PROGRAM DMXTest
VAR
	xConfigSet					: BOOL;
	xStatTestInProgress			: BOOL;
	xDMXSeqTestInProgressOnce	: BOOL;
	xDMXSeqTestInProgressTwice	: BOOL;
	xDMXSeqTestInProgressOnceDC	: BOOL;
	uiCounter2					: UINT;
	uiCounter3					: UINT;
	uiCounter4					: UINT;
	uiCounter5					: UINT;
	uiCounter6					: UINT;
	uiCounter7					: UINT;
	uiCounter8					: UINT;
	uiCounter9					: UINT;
	uiDedicatedRcvdRTIndex		: UINT;
	uiContinuousRTIndex			: UINT;
	
	uiForLoopCfgIndex			: UINT;
//	uiForLoopCtrlWriteIndex		: UINT;
//	uiForLoopCtrlWriteIndex2	: UINT;	
	uiLoopExpctdIndex			: UINT;
	uiForLoopClearExpctd		: UINT;
	uiLoopRcvIndex				: UINT;
	uiByteIndex					: UINT;
	iForLoopRecipeFindMin		: INT;
	iForLoopRecipeFindMax		: INT;
	iForLoopRecipeFindMax1		: INT;
	iForLoopRecipeMin			: INT;
	uiForLoopRecipe				: UINT;
	uiLoopIterDMXDUTArraySeq	: UINT;
	uiLoopIterDMXDUTArrayM		: UINT;
	uiLoopIterDUTArray24V		: UINT;
	uiLoopIterDUTArrayGND		: UINT;
	uiLoopIterTestArrSeq		: UINT;
	uiLoopIterTestArrM			: UINT;
	uiLoopIterTestArr24V		: UINT;
	uiLoopIterTestArrGND		: UINT;	
	iCompareStaticSM			: INT;
	iCompareSeq					: ARRAY[0..ENUM_SeqSM.Twice] OF INT;
	iParseFile					: INT;
	iSetConfig					: INT;
	iSetExpctdBufferSM			: INT;
	iReindexExpctedBufferSM		: INT;
	rt_RunStaticTest			: R_TRIG;
	rt_RunSeqTestOnce			: R_TRIG;
	rt_RunSeqTestOnceDC			: R_TRIG;
	rt_RunSeqTestTwice			: R_TRIG;
	rt_ResetTest				: R_TRIG;
	rt_ResetTestSeq				: R_TRIG;
	rt_ResetTestSeqDC			: R_TRIG;
	r_tStaticTestDone			: R_TRIG;
	
	//Arrays (Refactor 30-09-21)
	arr_uiRecipeIndexTmp		: ARRAY[0..gc.uiDUTConfigCountSplit] OF UINT;
 	arruiDMXChDUTTmp			: ARRAY[0..gc.uiDUTConfigCountSplit] OF UINT;
	arrsDUTChTypeTmp			: ARRAY[0..gc.uiDUTConfigCountSplit] OF STRING[3];	
	arr_uiRecipeIndex			: ARRAY[0..gc.uiDUTConfigCountSplit] OF UINT;
 	arruiDMXChDUT				: ARRAY[0..gc.uiDUTConfigCountSplit] OF UINT;
	arrsDUTChType				: ARRAY[0..gc.uiDUTConfigCountSplit] OF STRING[3];
	xFileImported				: BOOL;
	arr_usiRecipeSettingTmp		: ARRAY[0..gc.uiMaxNrOfDMXChannel] OF USINT;
	arr_usiRecipeSetting		: ARRAY[0..gc.uiMaxNrOfDMXChannel] OF USINT;






	
		
	arrxRcvdBufferPNP24V		: ARRAY[0..gc.uiMaxNrDMXTestCh] OF BOOL;
	arrxRcvdBufferNPN24V		: ARRAY[0..gc.uiMaxNrDMXTestCh] OF BOOL;
	arrxRcvdBufferPNPGND		: ARRAY[0..gc.uiMaxNrDMXTestCh] OF BOOL;
	arrxRcvdBufferNPNGND		: ARRAY[0..gc.uiMaxNrDMXTestCh] OF BOOL;
	
	arrxRcvdBufferPNPSeq		: ARRAY[0..gc.uiMaxNrDMXTestCh] OF BOOL;
	arrxRcvdBufferNPNSeq		: ARRAY[0..gc.uiMaxNrDMXTestCh] OF BOOL;	
	arrxRcvdBufferPNPMotor		: ARRAY[0..gc.uiMaxNrDMXTestCh] OF BOOL;
	arrxRcvdBufferNPNMotor		: ARRAY[0..gc.uiMaxNrDMXTestCh] OF BOOL;
	
	arrxExpctdPNP				: ARRAY[0..gc.uiMaxNrOfDMXChannel] OF BOOL; //What is expected based on the recipe file
	arrxExpctdNPN				: ARRAY[0..gc.uiMaxNrOfDMXChannel] OF BOOL; //What is expected based on the recipe file
	arrxExpctdTmpPNP			: ARRAY[0..gc.uiMaxNrOfDMXChannel] OF BOOL; //What is expected based on the recipe file, reindexed from DUT (usually 0)
	arrxExpctdTmpNPN			: ARRAY[0..gc.uiMaxNrOfDMXChannel] OF BOOL; //What is expected based on the recipe file, reindexed from DUT (usually 0)
	arrxExpctdTmpPNP24V			: ARRAY[0..gc.uiMaxNrDMXTestCh] OF BOOL; //What is expected based on the recipe file, reindexed from DUT (usually 0)
	arrxExpctdTmpNPN24V			: ARRAY[0..gc.uiMaxNrDMXTestCh] OF BOOL; //What is expected based on the recipe file, reindexed from DUT (usually 0)
	arrxExpctdTmpPNPGND			: ARRAY[0..gc.uiMaxNrDMXTestCh] OF BOOL; //What is expected based on the recipe file, reindexed from DUT (usually 0)
	arrxExpctdTmpNPNGND			: ARRAY[0..gc.uiMaxNrDMXTestCh] OF BOOL; //What is expected based on the recipe file, reindexed from DUT (usually 0)

	arrxExpctdTmpPNPSeqDMX		: ARRAY[0..gc.uiMaxNrDMXTestCh] OF BOOL; //What is expected based on the recipe file, reindexed from DUT (usually 0)
	arrxExpctdTmpNPNSeqDMX		: ARRAY[0..gc.uiMaxNrDMXTestCh] OF BOOL; //What is expected based on the recipe file, reindexed from DUT (usually 0)
	arrxExpctdTmpPNPSeqDC		: ARRAY[0..gc.uiMaxNrDMXTestCh] OF BOOL; //What is expected based on the recipe file, reindexed from DUT (usually 0)
	arrxExpctdTmpNPNSeqDC		: ARRAY[0..gc.uiMaxNrDMXTestCh] OF BOOL; //What is expected based on the recipe file, reindexed from DUT (usually 0)

	arrxExpctdTmpPNPSeq			: ARRAY[0..gc.uiMaxNrOfDMXChannel] OF BOOL; //What is expected based on the recipe file, reindexed from DUT (usually 0)
	arrxExpctdTmpNPNSeq			: ARRAY[0..gc.uiMaxNrOfDMXChannel] OF BOOL; //What is expected based on the recipe file, reindexed from DUT (usually 0)
	arrxExpctdTmpPNPMotor		: ARRAY[0..gc.uiMaxNrOfDMXChannel] OF BOOL; //What is expected based on the recipe file, reindexed from DUT (usually 0)
	arrxExpctdTmpNPNMotor		: ARRAY[0..gc.uiMaxNrOfDMXChannel] OF BOOL; //What is expected based on the recipe file, reindexed from DUT (usually 0)
	
	arrxExpctdMaskPNPSeq		: ARRAY[0..gc.uiMaxNrOfDMXChannel] OF BOOL; //Copy the contents of hardware buffer 
	arrxExpctdMaskNPNSeq		: ARRAY[0..gc.uiMaxNrOfDMXChannel] OF BOOL; //Copy the contents of hardware buffer 
	arr_diTestStaticPNP24V		: ARRAY[0..gc.uiMaxNrDMXTestCh] OF DINT;
	arr_diTestStaticNPN24V		: ARRAY[0..gc.uiMaxNrDMXTestCh] OF DINT;
	arr_diTestStaticPNPGND		: ARRAY[0..gc.uiMaxNrDMXTestCh] OF DINT;
	arr_diTestStaticNPNGND		: ARRAY[0..gc.uiMaxNrDMXTestCh] OF DINT;
	arr_diTestPNPSeqOnceLine			: ARRAY[0..gc.uiMaxNrDMXTestCh] OF DINT;
	arr_diTestPNPSeqOnceLineTmp			: ARRAY[0..gc.uiMaxNrDMXTestCh] OF DINT;
	arr_diTestNPNSeqOnceLine			: ARRAY[0..gc.uiMaxNrDMXTestCh] OF DINT;
	arr_diTestNPNSeqOnceLineTmp			: ARRAY[0..gc.uiMaxNrDMXTestCh] OF DINT;

	arr_udiMEMCPYPNPSeqOnceRcvdTmp		: ARRAY[0..gc.uiMaxNrDMXTestCh] OF UDINT;
	arr_udiMEMCPYNPNSeqOnceRcvdTmp		: ARRAY[0..gc.uiMaxNrDMXTestCh] OF UDINT;
			
	diTestStaticPNP24V				: DINT;
	diTestStaticNPN24V				: DINT;
	diTestStaticPNPGND				: DINT;	
	diTestStaticNPNGND				: DINT;
	
	diTestPNPSeqOnceComplete		: DINT;

	arrdiTestPNPSeqOnceComplete		: ARRAY[0..gc.uiMaxNrDMXTestCh] OF DINT;
	arrdiTestPNPSeqOnceCompleteTmp	: ARRAY[0..gc.uiMaxNrDMXTestCh] OF DINT;

	arrdiTestNPNSeqOnceComplete		: ARRAY[0..gc.uiMaxNrDMXTestCh] OF DINT;
	arrdiTestNPNSeqOnceCompleteTmp	: ARRAY[0..gc.uiMaxNrDMXTestCh] OF DINT;

	arrdiTestNPNSeqOnceCompleteProblemIndex		: ARRAY[0..gc.uiMaxNrDMXTestCh] OF DINT;
	
	arrudiStaticCopyResultPNP24V	: ARRAY[0..gc.uiMaxNrOfDMXChannel] OF UDINT;
	arrudiStaticCopyResultNPN24V	: ARRAY[0..gc.uiMaxNrOfDMXChannel] OF UDINT;
	arrudiStaticCopyResultPNPGND	: ARRAY[0..gc.uiMaxNrOfDMXChannel] OF UDINT;
	arrudiStaticCopyResultNPNGND	: ARRAY[0..gc.uiMaxNrOfDMXChannel] OF UDINT;	

	arr_diTestPNPMotorDir1		: ARRAY[0..gc.uiMaxNrDMXTestCh] OF DINT;
	arr_diTestNPNMotorDir1		: ARRAY[0..gc.uiMaxNrDMXTestCh] OF DINT;
	arr_diTestPNPMotorDir2		: ARRAY[0..gc.uiMaxNrDMXTestCh] OF DINT;
	arr_diTestNPNMotorDir2		: ARRAY[0..gc.uiMaxNrDMXTestCh] OF DINT;

	
	
	diCompTestResult			: DINT;
	diCompTestResultTemp		: DINT;
	diTestResultStaticPNP		: DINT;
	diTestResultStaticNPN		: DINT;	

	arrVisu_diTestResult		: ARRAY[0..gc.uiMaxNrDMXTestCh] OF DINT;
	uiVisuIndex					: UINT;
	tonReadWait					: TON;
	tonConvert					: TON;
	tonWriteCopyWait			: TON;
	tonTestIterGap				: TON;
	tTestTime					: TIME;
	tWriteWaitTime				: TIME;
	r_tSetConfig				: R_TRIG;
	uiRecipeIndexRcv			: UINT;
	uiMinRecipeIndex			: UINT;
	uiMaxRecipeIndex			: UINT;
	cuiMinDUTIndex				: UINT	:= 0; // Constant
	uiMaxRecipeIndexTemp		: UINT;
	arruiMotorTestIndices		: ARRAY[0..gc.uiMaxNrOfDMXChannel] OF UINT;
	arruiMotorTestIndicesTmp	: ARRAY[0..gc.uiMaxNrOfDMXChannel] OF UINT;
	arruiSeqTestIndices			: ARRAY[0..gc.uiMaxNrOfDMXChannel] OF UINT;
	arruiSeqTestIndicesTmp		: ARRAY[0..gc.uiMaxNrOfDMXChannel] OF UINT;
	
	arruiSeqTestIndicesDMX			: ARRAY[0..gc.uiMaxNrDMXTestCh] OF UINT;
	arruiSeqTestIndicesDMXSW		: ARRAY[0..gc.uiMaxNrDMXTestCh] OF UINT;
	arruiSeqTestIndicesDMXTmp		: ARRAY[0..gc.uiMaxNrDMXTestCh] OF UINT;
	
	arruiSeqTestIndicesDC			: ARRAY[0..gc.uiMaxNrDMXTestCh] OF UINT;
	arruiSeqTestIndicesDCTmp		: ARRAY[0..gc.uiMaxNrDMXTestCh] OF UINT;	
	
	arrui24VTestIndices			: ARRAY[0..gc.uiMaxNrOfDMXChannel] OF UINT;
	arrui24VTestIndicesTmp		: ARRAY[0..gc.uiMaxNrOfDMXChannel] OF UINT;
	arruiGNDTestIndices			: ARRAY[0..gc.uiMaxNrOfDMXChannel] OF UINT;
	arruiGNDTestIndicesTmp		: ARRAY[0..gc.uiMaxNrOfDMXChannel] OF UINT;
	udiMemCpyResultPNP			: UDINT;
	udiMemCpyResultDMX			: UDINT;	
	r_tSetExpectedBuff			: R_TRIG;
	r_tExpectedBufferSet		: R_TRIG;
	uiLoopExpctdIndexRead		: UINT;
	uiLoopExpctdIndexWrite		: UINT;
	xTestBoolDelete				: BOOL;
	uiForLoopZeroStorageArray	: UINT;
	
	//For DUT Config
	r_tSetDUTVal				: R_TRIG;
	usiDUTVal					: USINT;
	uiForLoopDUTIter			: UINT;
	iSetDUTSM					: INT;
	
	//For 'Invert Recipe Settings'
	uiStartingIndex				: UINT;
	uiEndingIndex				: UINT;
	uiRecipeInvertIter			: UINT;
	R_TInvertRecipe				: R_TRIG;
	iInvertRecipeSM				: INT;
END_VAR

SeqTestOnce();
//SeqTestTwice();
//SeqTestOnceDC();
InvertRecipeSettings();
rt_RunStaticTest();
rt_ResetTest();
r_tSetConfig();//Set config when file is loaded; this condition happens when End-of-File (EOF) is reached; set by HMI button
r_tSetExpectedBuff(CLK:=r_tSetConfig.Q);
r_tExpectedBufferSet();
r_tStaticTestDone(CLK			:= (iCompareStaticSM = 110));
r_tSetDUTVal();
tonReadWait(PT		:= tTestTime);
tonConvert(PT		:= tTestTime);
tonWriteCopyWait(PT	:= tWriteWaitTime);
tonTestIterGap(PT	:= tTestTime);
tTestTime			:= T#80MS;
//just an example one
tWriteWaitTime		:= T#10MS; // same as the tOffDelay set to the input debounce FB
//DMX DUT Channels, Software 0-255 
//DMX Config Channels, Software, 256-511
//DMX DUT Channels, Hardware 1-256
//DMX Config Channels, Hardware, 257-512

//Interface Link - continued - DMXTest Local Vars

//"Config Complete" Expctd Buffer, and "Config Complete" Received Buffer; then Global Comparison is like 'masking' all but one channel at a time;

CASE iParseFile OF

0:
IF P_TextModeRead.r_tFileChg.Q THEN
	xFileImported		:= FALSE;	
	iParseFile			:= 5;
END_IF

5:
IF P_TextModeRead.fbFileGets.bEOF THEN
	uiForLoopRecipe	:= 0; // Reset the iterator used in the next state of the SM
	iParseFile		:= 10;
END_IF
	
10://At first check for any recipe items specified in the file;
//Load the recipe data into respective arrays
//For recipe indices = 0 to 255, parse the file to read the recipe index, DMX channel, and channel type
FOR uiForLoopRecipe := 0 TO gc.uiDUTConfigCountSplit BY 1 DO
	//Read the Recipe Index
	arr_uiRecipeIndexTmp[uiForLoopRecipe]		:= STRING_TO_UINT(P_TextModeRead.database[uiForLoopRecipe,0]);
	//Read the DMX Channel for the DUT
	arruiDMXChDUTTmp[uiForLoopRecipe]			:= STRING_TO_UINT(P_TextModeRead.database[uiForLoopRecipe,1]);
	//Read the type of Channel on the DUT
	arrsDUTChTypeTmp[uiForLoopRecipe]			:= P_TextModeRead.database[uiForLoopRecipe,2];
END_FOR
//Stash the values from temp (inside FOR loop) to other arrays
arr_uiRecipeIndex	:= arr_uiRecipeIndexTmp;
arruiDMXChDUT		:= arruiDMXChDUTTmp;
arrsDUTChType		:= arrsDUTChTypeTmp;

//If the 'TextModeRead' re-enters 'Ready' state then advance this SM
IF P_TextModeRead.step = 0 THEN
	xFileImported		:= TRUE;
	iParseFile			:= 0;	
END_IF

END_CASE

CASE iSetConfig OF

//Don't look at the P_TextRead; evaluate on the arrays you just imported

0:
IF r_tSetConfig.Q THEN
	iSetConfig			:= 10;	
END_IF

10://Read the string that is loaded from file reader; pass value to DMX Function Block, at the appropriate Config index
//This is the setting to control the position of the 'config' relays on the tester
//Ensure that the declared arrays are sufficiently long to handle the max conceivable value (512 x 2, in this case?)
FOR uiForLoopRecipe := 0 TO gc.uiDUTConfigCountSplit BY 1 DO
	IF (arruiDMXChDUT[uiForLoopRecipe] <> 0) THEN
		//Set the config routing := NPN
		arr_usiRecipeSettingTmp[(uiForLoopRecipe+gc.uiChannelSplitCount)]	:= 255;
	ELSIF (arruiDMXChDUT[uiForLoopRecipe] = 0) THEN
		//Set the config routing := PNP
		arr_usiRecipeSettingTmp[(uiForLoopRecipe+gc.uiChannelSplitCount)]	:= 0;
	END_IF	
END_FOR
//Stash the values from temp (inside FOR loop) to other arrays
arr_usiRecipeSetting	:= arr_usiRecipeSettingTmp;

	iSetConfig			:= 20;	

20://Iterate over the config listings to create indices for what must be tested static (power, ground), and what must be tested sequentially (channels)
uiLoopIterDMXDUTArraySeq	:= 0;
uiLoopIterTestArrSeq		:= 0;
//Zero out the array that is copied to in the next state of the SM
FOR uiForLoopZeroStorageArray	:= 0 TO gc.uiMaxNrOfDMXChannel BY 1 DO
	arruiSeqTestIndicesTmp[uiForLoopZeroStorageArray]	:= 0;
END_FOR
//Stash the values from temp (inside FOR loop) to other arrays
arruiSeqTestIndices		:= arruiSeqTestIndicesTmp;
iSetConfig				:= 40;	

40:
//For any 'DMX'-type channels with an assigned channel # (from the recipe), then copy only those elements to another array
//These are elements that are tested sequentially - once - so this includes Dry Contacts but not Motors
REPEAT
	IF ((arrsDUTChType[uiLoopIterDMXDUTArraySeq] = 'DMX') OR (arrsDUTChType[uiLoopIterDMXDUTArraySeq] = '24V')) AND (arruiDMXChDUT[uiLoopIterDMXDUTArraySeq] <> 0) THEN
		MEMCPY(srcAddr:=ADR(arruiDMXChDUT[uiLoopIterDMXDUTArraySeq]),destAddr:=ADR(arruiSeqTestIndicesTmp[uiLoopIterDMXDUTArraySeq]),n:=SIZEOF(arruiDMXChDUT[uiLoopIterDMXDUTArraySeq])); //UINT = 4 bytes?
//		uiLoopIterTestArrSeq		:= uiLoopIterTestArrSeq+1;
	END_IF
	uiLoopIterDMXDUTArraySeq	:= uiLoopIterDMXDUTArraySeq+1;
UNTIL 
(uiLoopIterDMXDUTArraySeq = gc.uiMaxNrOfDMXChannel)
END_REPEAT
//Stash the values from temp (inside FOR loop) to other arrays
arruiSeqTestIndices		:= arruiSeqTestIndicesTmp;

iSetConfig					:= 50;	

50:
//Use different iterators - set them to 0 prior to use
uiLoopIterDMXDUTArrayM		:= 0;
uiLoopIterTestArrM			:= 0;
//Zero out the array that is copied to in the next state of the SM
FOR uiForLoopZeroStorageArray	:= 0 TO gc.uiMaxNrOfDMXChannel BY 1 DO
	arruiMotorTestIndicesTmp[uiForLoopZeroStorageArray]	:= 0;
END_FOR
//Stash the values from temp (inside FOR loop) to other arrays
arruiMotorTestIndices	:= arruiMotorTestIndicesTmp;

iSetConfig					:= 60;	

60:
//Motors - Type code "M" - must be tested both in the PNP & NPN inputs
//This array easily provides the indexing for which channels the motors are on
REPEAT
	IF (arrsDUTChType[uiLoopIterDMXDUTArrayM] = 'M') AND (arruiDMXChDUT[uiLoopIterDMXDUTArrayM] <> 0)  THEN
		MEMCPY(srcAddr:=ADR(arruiDMXChDUT[uiLoopIterDMXDUTArrayM]),destAddr:=ADR(arruiMotorTestIndicesTmp[uiLoopIterDMXDUTArrayM]),n:=SIZEOF(arruiDMXChDUT[uiLoopIterDMXDUTArrayM])); //UINT = 4 bytes?
//		uiLoopIterTestArrM		:= uiLoopIterTestArrM+1;
	END_IF
	uiLoopIterDMXDUTArrayM	:= uiLoopIterDMXDUTArrayM+1;
UNTIL 
(uiLoopIterDMXDUTArrayM = gc.uiMaxNrOfDMXChannel)
END_REPEAT
//Stash the values from temp (inside FOR loop) to other arrays
arruiMotorTestIndices	:= arruiMotorTestIndicesTmp;

iSetConfig		:= 70;

70:
//Use different iterators - set them to 0 prior to use
uiLoopIterDUTArray24V		:= 0;
uiLoopIterTestArr24V		:= 0;
//Zero out the array that is copied to in the next state of the SM
FOR uiForLoopZeroStorageArray	:= 0 TO gc.uiMaxNrOfDMXChannel BY 1 DO
	arrui24VTestIndicesTmp[uiForLoopZeroStorageArray]	:= 0;
END_FOR
//Stash the values from temp (inside FOR loop) to other arrays
arrui24VTestIndices		:= arrui24VTestIndicesTmp;

iSetConfig				:= 80;

80:
//24V - Type code "24V" - is tested per static config
//This array easily provides the indexing for which channels the 24V are on
REPEAT
	IF (arrsDUTChType[uiLoopIterDUTArray24V] = '24V') AND (arruiDMXChDUT[uiLoopIterDUTArray24V] = 0) THEN
		MEMCPY(srcAddr:=ADR(arr_uiRecipeIndex[uiLoopIterDUTArray24V]),destAddr:=ADR(arrui24VTestIndicesTmp[uiLoopIterDUTArray24V]),n:=SIZEOF(arr_uiRecipeIndex[uiLoopIterDUTArray24V])); //UINT = 2 bytes?
//		uiLoopIterTestArr24V	:= uiLoopIterTestArr24V +1;
	END_IF
	uiLoopIterDUTArray24V	:= uiLoopIterDUTArray24V+1;
UNTIL 
(uiLoopIterDUTArray24V = gc.uiDUTConfigCountSplit)
END_REPEAT
//Stash the values from temp (inside FOR loop) to other arrays
arrui24VTestIndices	:= arrui24VTestIndicesTmp;

iSetConfig		:= 90;

90://Clear Iterators for GND channel indexing
//Use different iterators - set them to 0 prior to use
uiLoopIterDUTArrayGND		:= 0;
uiLoopIterTestArrGND		:= 0;
//Zero out the array that is copied to in the next state of the SM
FOR uiForLoopZeroStorageArray	:= 0 TO gc.uiMaxNrOfDMXChannel BY 1 DO
	arruiGNDTestIndicesTmp[uiForLoopZeroStorageArray]	:= 0;
END_FOR
//Stash the values from temp (inside FOR loop) to other arrays
arruiGNDTestIndices		:= arruiGNDTestIndicesTmp;

iSetConfig				:= 100;

100:
//Ground - Type code "GND" - is tested per static config
//This array easily provides the indexing for which channels the 24V are on
REPEAT
	IF (arrsDUTChType[uiLoopIterDUTArrayGND] = 'GND') AND (arruiDMXChDUT[uiLoopIterDUTArrayGND] = 0) THEN
		MEMCPY(srcAddr:=ADR(arr_uiRecipeIndex[uiLoopIterDUTArrayGND]),destAddr:=ADR(arruiGNDTestIndicesTmp[uiLoopIterDUTArrayGND]),n:=SIZEOF(arr_uiRecipeIndex[uiLoopIterDUTArrayGND])); //UINT = 4 bytes?
//		uiLoopIterTestArrGND	:= uiLoopIterTestArrGND+1;
	END_IF
	uiLoopIterDUTArrayGND	:= uiLoopIterDUTArrayGND+1;
UNTIL 
(uiLoopIterDUTArrayGND = gc.uiDUTConfigCountSplit)
END_REPEAT
//Stash the values from temp (inside FOR loop) to other arrays
arruiGNDTestIndices	:= arruiGNDTestIndicesTmp;

iSetConfig				:= 110;

//Copy of state30
110://Iterate over the config listings to create indices for what must be tested static (power, ground), and what must be tested sequentially (channels)
uiLoopIterDMXDUTArraySeq		:= 0;
uiLoopIterTestArrSeq			:= 0;
//Zero out the array that is copied to in the next state of the SM
FOR uiForLoopZeroStorageArray	:= 0 TO gc.uiMaxNrOfDMXChannel BY 1 DO
	arruiSeqTestIndicesDMXTmp[uiForLoopZeroStorageArray]	:= 0;
	arruiSeqTestIndicesDMXSW[uiForLoopZeroStorageArray]		:= 0;
END_FOR
//Stash the values from temp (inside FOR loop) to other arrays
arruiSeqTestIndicesDMX			:= arruiSeqTestIndicesDMXTmp;
iSetConfig						:= 120;	

120://Effectively a copy of state40
//For any 'DMX'-type channels with an assigned channel # (from the recipe), then copy only those elements to another array
//These are elements that are tested sequentially - once - so this includes Dry Contacts but not Motors
REPEAT
	IF (arrsDUTChType[uiLoopIterDMXDUTArraySeq] = 'DMX') AND (arruiDMXChDUT[uiLoopIterDMXDUTArraySeq] <> 0) THEN
		MEMCPY(srcAddr:=ADR(arruiDMXChDUT[uiLoopIterDMXDUTArraySeq]),destAddr:=ADR(arruiSeqTestIndicesDMXTmp[uiLoopIterDMXDUTArraySeq]),n:=SIZEOF(arr_uiRecipeIndex[uiLoopIterDUTArrayGND])); //UINT = 4 bytes?
//		uiLoopIterTestArrSeq		:= uiLoopIterTestArrSeq+1;
	END_IF
	uiLoopIterDMXDUTArraySeq		:= uiLoopIterDMXDUTArraySeq+1;
UNTIL 
(uiLoopIterDMXDUTArraySeq = gc.uiMaxNrOfDMXChannel)
END_REPEAT
//Stash the values from temp (inside FOR loop) to other arrays
arruiSeqTestIndicesDMX				:= arruiSeqTestIndicesDMXTmp;

//Set the recipe addresses one lower for 'SW'-Software-because software indexes from 0, not 1
FOR uiCounter8	:= 0 TO gc.uiMaxNrDMXTestCh BY 1 DO
	IF arruiSeqTestIndicesDMX[uiCounter8] <> 0 THEN
		arruiSeqTestIndicesDMXSW[uiCounter8]	:= arruiSeqTestIndicesDMX[uiCounter8] - 1;	
	END_IF
END_FOR

iSetConfig							:= 130;	

//Copy of state30
130://Iterate over the config listings to create indices for what must be tested static (power, ground), and what must be tested sequentially (channels)
uiLoopIterDMXDUTArraySeq		:= 0;
uiLoopIterTestArrSeq			:= 0;
//Zero out the array that is copied to in the next state of the SM
FOR uiForLoopZeroStorageArray	:= 0 TO gc.uiMaxNrOfDMXChannel BY 1 DO
	arruiSeqTestIndicesDCTmp[uiForLoopZeroStorageArray]	:= 0;
END_FOR
//Stash the values from temp (inside FOR loop) to other arrays
arruiSeqTestIndicesDC			:= arruiSeqTestIndicesDCTmp;
iSetConfig						:= 140;	

140:
//For any 'DMX'-type channels with an assigned channel # (from the recipe), then copy only those elements to another array
//These are elements that are tested sequentially - once - so this includes Dry Contacts but not Motors
REPEAT
	IF (arrsDUTChType[uiLoopIterDMXDUTArraySeq] = '24V') AND (arruiDMXChDUT[uiLoopIterDMXDUTArraySeq] <> 0) THEN
		MEMCPY(srcAddr:=ADR(arruiDMXChDUT[uiLoopIterDMXDUTArraySeq]),destAddr:=ADR(arruiSeqTestIndicesDCTmp[uiLoopIterDMXDUTArraySeq]),n:=SIZEOF(arruiDMXChDUT[uiLoopIterDMXDUTArraySeq])); //UINT = 4 bytes?
//		uiLoopIterTestArrSeq		:= uiLoopIterTestArrSeq+1;
	END_IF
	uiLoopIterDMXDUTArraySeq		:= uiLoopIterDMXDUTArraySeq+1;
UNTIL 
(uiLoopIterDMXDUTArraySeq = gc.uiMaxNrOfDMXChannel)
END_REPEAT
//Stash the values from temp (inside FOR loop) to other arrays
arruiSeqTestIndicesDC				:= arruiSeqTestIndicesDCTmp;

iSetConfig							:= 0;	

END_CASE


//Set the config of the 'routing' channels
IF r_tSetConfig.Q THEN
	g_ast.DMXHWOut	:= g_ast.DMXPhysOut;
//	xConfigSet		:= TRUE;
END_IF


// For manual setting of channels from the Visualization - NOTE! This stamps over any other values set for the lower 256 channels (DUT)
CASE iSetDUTSM OF
	
0:
IF r_tSetDUTVal.Q THEN
	iSetDUTSM		:= 10;
END_IF

10:
FOR uiForLoopDUTIter := 0 TO gc.uiDUTConfigCountSplit BY 1 DO
	g_ast.DMXHWOut[uiForLoopDUTIter] 	:= usiDUTVal;
END_FOR
//g_ast.DMXHWOut					:= g_ast.DMXPhysOut;

IF NOT r_tSetDUTVal.Q THEN
	iSetDUTSM	:= 0;
END_IF

END_CASE


CASE iSetExpctdBufferSM OF
	
0://If there is a trigger to set the test config, create a new 'Expctd' buffer
IF r_tSetExpectedBuff.Q THEN
	r_tExpectedBufferSet.CLK	:= FALSE;
	//Clear the existing buffers
	FOR uiForLoopClearExpctd := 0 TO gc.uiMaxNrOfDMXChannel BY 1 DO
		arrxExpctdPNP[uiForLoopClearExpctd]	:= 0;
		arrxExpctdNPN[uiForLoopClearExpctd]	:= 0;
	END_FOR
	iSetExpctdBufferSM			:= 10;
END_IF

10: // Set Expected Buffers per Recipe Files
FOR uiLoopExpctdIndex := 0 TO gc.uiMaxNrOfDMXChannel BY 1 DO
	IF (arr_usiRecipeSetting[uiLoopExpctdIndex] <= 127) THEN
		arrxExpctdPNP[arr_uiRecipeIndex[uiLoopExpctdIndex]]		:= TRUE; 
		arrxExpctdNPN[arr_uiRecipeIndex[uiLoopExpctdIndex]]		:= FALSE;
	ELSIF (arr_usiRecipeSetting[uiLoopExpctdIndex] > 127) THEN
		arrxExpctdPNP[arr_uiRecipeIndex[uiLoopExpctdIndex]]		:= FALSE;
		arrxExpctdNPN[arr_uiRecipeIndex[uiLoopExpctdIndex]]		:= TRUE; 
	END_IF
	//Zero out Expected, type-specific index buffers
	arrxExpctdTmpPNP24V[uiLoopExpctdIndex] 					:= 0;
	arrxExpctdTmpNPN24V[uiLoopExpctdIndex] 					:= 0;
	arrxExpctdTmpPNPGND[uiLoopExpctdIndex] 					:= 0;
	arrxExpctdTmpNPNGND[uiLoopExpctdIndex] 					:= 0;
END_FOR

r_tExpectedBufferSet.CLK	:= TRUE;
iSetExpctdBufferSM			:= 0;

END_CASE

CASE iReindexExpctedBufferSM OF
	
0:
IF r_tExpectedBufferSet.Q THEN
	iReindexExpctedBufferSM	:= 10;
END_IF

10://Copy the contents of Expected Buffer to a different Buffer, starting at array address 0 - only the channels that have a hardware input index
MEMCPY(srcAddr:=ADR(arrxExpctdPNP[gc.uiChannelSplitCount]),destAddr:=ADR(arrxExpctdTmpPNP[cuiMinDUTIndex]),n:=gc.uiChannelsUT);
MEMCPY(srcAddr:=ADR(arrxExpctdNPN[gc.uiChannelSplitCount]),destAddr:=ADR(arrxExpctdTmpNPN[cuiMinDUTIndex]),n:=gc.uiChannelsUT);

iReindexExpctedBufferSM	:= 20;

20:
//And create the comparison Expected Buffer for Static Test - 24V & GND indices
FOR uiCounter5 := 0 TO gc.uiMaxNrDMXTestCh BY 1 DO
	IF arrui24VTestIndices[uiCounter5] <> 0 THEN	
		MEMCPY(srcAddr:=ADR(arrxExpctdTmpPNP[arrui24VTestIndices[uiCounter5]]),destAddr:=ADR(arrxExpctdTmpPNP24V[arrui24VTestIndices[uiCounter5]]),n:=SIZEOF(arrxExpctdTmpPNP[arrui24VTestIndices[uiCounter5]])); //bytes
		MEMCPY(srcAddr:=ADR(arrxExpctdTmpNPN[arrui24VTestIndices[uiCounter5]]),destAddr:=ADR(arrxExpctdTmpNPN24V[arrui24VTestIndices[uiCounter5]]),n:=SIZEOF(arrxExpctdTmpNPN[arrui24VTestIndices[uiCounter5]])); //bytes
	END_IF
	
	IF arruiGNDTestIndices[uiCounter5] <> 0 THEN	
		MEMCPY(srcAddr:=ADR(arrxExpctdTmpPNP[arruiGNDTestIndices[uiCounter5]]),destAddr:=ADR(arrxExpctdTmpPNPGND[arruiGNDTestIndices[uiCounter5]]),n:=SIZEOF(arrxExpctdTmpPNP[arruiGNDTestIndices[uiCounter5]])); //bytes
		MEMCPY(srcAddr:=ADR(arrxExpctdTmpNPN[arruiGNDTestIndices[uiCounter5]]),destAddr:=ADR(arrxExpctdTmpNPNGND[arruiGNDTestIndices[uiCounter5]]),n:=SIZEOF(arrxExpctdTmpNPN[arruiGNDTestIndices[uiCounter5]])); //bytes
	END_IF	
END_FOR

iReindexExpctedBufferSM	:= 0;

END_CASE


CASE iCompareStaticSM OF
	
0: // If test is triggered by user
IF rt_RunStaticTest.Q THEN
	xStatTestInProgress						:= TRUE;
	uiLoopRcvIndex							:= cuiMinDUTIndex; 
	iCompareStaticSM						:= 10;
END_IF

10: // Zero out all comparison buffers before each comparison
//IF (uiLoopRcvIndex=0) THEN
	IF xStatTestInProgress THEN
		//by default, Counter = 0 at the first initialization; it is reset at the end of this State Machine
		//Clear Storage Buffers pre-test to ensure no old data interferes with current test
		FOR uiCounter4 := 0 TO gc.uiDUTConfigCountSplit BY 1 DO
			arrxRcvdBufferPNP24V[uiCounter4]	:= 0;		
			arrxRcvdBufferNPN24V[uiCounter4]	:= 0;		
			arrxRcvdBufferPNPGND[uiCounter4]	:= 0;		
			arrxRcvdBufferNPNGND[uiCounter4]	:= 0;
			gFB.arrFB_DMX[uiCounter4].I.xCmdOff	:= TRUE;		
//			g_ast.DMX[uiCounter4].IQ.xCmdOff	:= TRUE;	
		END_FOR
	iCompareStaticSM				:= 20;
	END_IF
(*
ELSIF (uiLoopRcvIndex>0) THEN
	IF xStatTestInProgress AND tonTestIterGap.Q THEN
		tonTestIterGap.IN	:= FALSE;
		//by default, Counter = 0 at the first initialization; it is reset at the end of this State Machine
		//Clear Storage Buffers pre-test to ensure no old data interferes with current test
		FOR uiCounter4 := 0 TO gc.uiDUTConfigCountSplit BY 1 DO
			arrxRcvdBufferPNP24V[uiCounter4]	:= 0;		
			arrxRcvdBufferNPN24V[uiCounter4]	:= 0;		
			arrxRcvdBufferPNPGND[uiCounter4]	:= 0;		
			arrxRcvdBufferNPNGND[uiCounter4]	:= 0;		
		END_FOR
	iCompareStaticSM				:= 30; // don't write the hardware value (skip 20)
	END_IF
END_IF
*)
	
20:	
//write 'hardware-clear' state 
g_ast.DMXHWOut					:= g_ast.DMXPhysOut;
iCompareStaticSM				:= 30;

30: //Set the Expected Mask & write data to controller
(*
IF uiLoopRcvIndex <> 0 THEN
//	g_ast.DMX[uiLoopRcvIndex].IQ.xCmdOn			:= TRUE;
	FOR uiCounter3 := cuiMinDUTIndex TO gc.uiMaxNrDMXTestCh BY 1 DO
		IF uiCounter3 <> uiLoopRcvIndex THEN
			g_ast.DMX[uiCounter3].IQ.xCmdOff	:= TRUE;	
		END_IF
	END_FOR
	iCompareStaticSM		:= 40;
ELSE //uiLoopRcvIndex = 0
	*)
tonWriteCopyWait.IN		:= TRUE;
iCompareStaticSM		:= 50;
//END_IF

40:
//Write DMX channels
(*
g_ast.DMXHWOut			:= g_ast.DMXPhysOut;
tonWriteCopyWait.IN		:= TRUE;
iCompareStaticSM		:= 50;
*)

50:
IF tonWriteCopyWait.Q THEN
	tonWriteCopyWait.IN	:= FALSE;
	iCompareStaticSM	:= 60;
END_IF

60:
FOR uiCounter4 := 0 TO gc.uiMaxNrDMXTestCh BY 1 DO

//IF there is an index for a '24V' element, then copy that element's value to a new pair of arrays, for 'Received'

	IF arrui24VTestIndices[uiCounter4] <> 0 THEN

		arrudiStaticCopyResultPNP24V[arrui24VTestIndices[uiCounter4]]	:= MEMCPY(srcAddr:=ADR(g_ast.arrInputPNP[arrui24VTestIndices[uiCounter4]]),destAddr:=ADR(arrxRcvdBufferPNP24V[arrui24VTestIndices[uiCounter4]]),n:=SIZEOF(g_ast.arrInputPNP[arrui24VTestIndices[uiCounter4]])); //bytes
		arrudiStaticCopyResultNPN24V[arrui24VTestIndices[uiCounter4]]	:= MEMCPY(srcAddr:=ADR(g_ast.arrInputNPN[arrui24VTestIndices[uiCounter4]]),destAddr:=ADR(arrxRcvdBufferNPN24V[arrui24VTestIndices[uiCounter4]]),n:=SIZEOF(g_ast.arrInputNPN[arrui24VTestIndices[uiCounter4]])); //bytes)

	END_IF

//IF there is an index for a 'GND' element, then copy that element's value to a new pair of arrays, for 'Received'

	IF arruiGNDTestIndices[uiCounter4] <> 0 THEN

		arrudiStaticCopyResultPNPGND[arruiGNDTestIndices[uiCounter4]]	:= MEMCPY(srcAddr:=ADR(g_ast.arrInputPNP[arruiGNDTestIndices[uiCounter4]]),destAddr:=ADR(arrxRcvdBufferPNPGND[arruiGNDTestIndices[uiCounter4]]),n:=SIZEOF(g_ast.arrInputPNP[arruiGNDTestIndices[uiCounter4]])); //bytes
		arrudiStaticCopyResultNPNGND[arruiGNDTestIndices[uiCounter4]]	:= MEMCPY(srcAddr:=ADR(g_ast.arrInputNPN[arruiGNDTestIndices[uiCounter4]]),destAddr:=ADR(arrxRcvdBufferNPNGND[arruiGNDTestIndices[uiCounter4]]),n:=SIZEOF(g_ast.arrInputNPN[arruiGNDTestIndices[uiCounter4]])); //bytes)
	
	END_IF
	
END_FOR

iCompareStaticSM			:= 70;

70:
tonReadWait.IN				:= TRUE;
iCompareStaticSM			:= 80;

80: // if wait completed, set the bit for conversion high
//Conversion Function call
IF tonReadWait.Q THEN
	tonReadWait.IN					:= FALSE;
	iCompareStaticSM				:= 90;
END_IF

90:
//Run Comparos
//Individual Channels comparison
FOR uiCounter6	:= 0 TO gc.uiMaxNrDMXTestCh BY 1 DO 
	arr_diTestStaticPNP24V[uiCounter6]		:= MEMCMP(pBuf1:=ADR(arrxExpctdTmpPNP24V[uiCounter6]),pBuf2:=ADR(arrxRcvdBufferPNP24V[uiCounter6]),n:=SIZEOF(arrxExpctdTmpPNP24V[uiCounter6]));
	arr_diTestStaticNPN24V[uiCounter6]		:= MEMCMP(pBuf1:=ADR(arrxExpctdTmpNPN24V[uiCounter6]),pBuf2:=ADR(arrxRcvdBufferNPN24V[uiCounter6]),n:=SIZEOF(arrxExpctdTmpNPN24V[uiCounter6]));
	arr_diTestStaticPNPGND[uiCounter6]		:= MEMCMP(pBuf1:=ADR(arrxExpctdTmpPNPGND[uiCounter6]),pBuf2:=ADR(arrxRcvdBufferPNPGND[uiCounter6]),n:=SIZEOF(arrxExpctdTmpPNPGND[uiCounter6]));
	arr_diTestStaticNPNGND[uiCounter6]		:= MEMCMP(pBuf1:=ADR(arrxExpctdTmpNPNGND[uiCounter6]),pBuf2:=ADR(arrxRcvdBufferNPNGND[uiCounter6]),n:=SIZEOF(arrxExpctdTmpNPNGND[uiCounter6]));
END_FOR

//Complete Buffer
diTestStaticPNP24V		:= MEMCMP(pBuf1:=ADR(arrxExpctdTmpPNP24V[cuiMinDUTIndex]),pBuf2:=ADR(arrxRcvdBufferPNP24V[cuiMinDUTIndex]),n:=gc.uiChannelsUT);
diTestStaticNPN24V		:= MEMCMP(pBuf1:=ADR(arrxExpctdTmpNPN24V[cuiMinDUTIndex]),pBuf2:=ADR(arrxRcvdBufferNPN24V[cuiMinDUTIndex]),n:=gc.uiChannelsUT);
diTestStaticPNPGND		:= MEMCMP(pBuf1:=ADR(arrxExpctdTmpPNPGND[cuiMinDUTIndex]),pBuf2:=ADR(arrxRcvdBufferPNPGND[cuiMinDUTIndex]),n:=gc.uiChannelsUT);
diTestStaticNPNGND		:= MEMCMP(pBuf1:=ADR(arrxExpctdTmpNPNGND[cuiMinDUTIndex]),pBuf2:=ADR(arrxRcvdBufferNPNGND[cuiMinDUTIndex]),n:=gc.uiChannelsUT);

iCompareStaticSM				:= 105;

(*
100: // If counter is equal to the max # of test channels, reset it; turn off the DMX channels that were turned on in the course of the test
IF (uiLoopRcvIndex = gc.uiMaxNrDMXTestCh) THEN
	rt_RunStaticTest.CLK			:= TRUE;
	iCompareStaticSM				:= 110;
ELSE
	uiLoopRcvIndex				:= uiLoopRcvIndex +1;
	//Next iteration
	tonTestIterGap.IN			:= TRUE;
	iCompareStaticSM			:= 10;
 (*iCounter <> gc.usiMaxNrOfChannels*)
END_IF
*)

105:
//Retrieving the discrepant indices for display on HMI
FOR uiVisuIndex := 0 TO gc.uiMaxNrDMXTestCh BY 1 DO
	IF (arr_diTestStaticPNP24V[uiVisuIndex] <> 0) THEN
		arrVisu_diTestResult[uiVisuIndex]	:= uiVisuIndex;	
	ELSIF (arr_diTestStaticNPNGND[uiVisuIndex] <> 0) THEN
		arrVisu_diTestResult[uiVisuIndex]	:= uiVisuIndex;	
	END_IF
END_FOR

iCompareStaticSM				:= 110;
	
110:
xStatTestInProgress				:= FALSE;
iCompareStaticSM				:= 120;

120:
IF rt_ResetTest.Q AND NOT rt_RunStaticTest.Q THEN
	FOR uiCounter2 := 0 TO gc.uiMaxNrDMXTestCh BY 1 DO 
		arr_diTestStaticPNP24V[uiCounter2]		:= 0;
		arr_diTestStaticNPN24V[uiCounter2]		:= 0;
		arr_diTestStaticPNPGND[uiCounter2]		:= 0;
		arr_diTestStaticNPNGND[uiCounter2]		:= 0;
	END_FOR
	diCompTestResult							:= 0;
	iCompareStaticSM							:= 0; (* reset to beginning *)
END_IF

END_CASE


//Linked to the Visualization Table
//FOR uiVisuIndex := 0 TO gc.uiMaxNrDMXTestCh BY 1 DO
	//	arrVisu_diTestResult[0,uiVisuIndex]	:= g_ast.DMXHWOut[uiVisuIndex]; //Sent
	//	arrVisu_diTestResult[1,uiVisuIndex]	:= arrbySclPNP[uiVisuIndex]; //Received
	//	arrVisu_diTestResult[2,uiVisuIndex]	:= arr_diTestResultPNP[uiVisuIndex]; //Result of Comparison
	//	arrVisu_diTestResult[3,uiVisuIndex]	:= arr_diTestResultNPN[uiVisuIndex]; //Result of Comparison
//END_FOR



//IF diCompTestResultTemp = -1 OR diCompTestResultTemp = 1 THEN
//	diCompTestResult	:= diCompTestResultTemp;
//END_IF

ACTION InvertRecipeSettings:
R_TInvertRecipe();

CASE iInvertRecipeSM OF
	
0:
IF R_TInvertRecipe.Q THEN
	iInvertRecipeSM		:= 10;
END_IF

10:
FOR uiRecipeInvertIter := uiStartingIndex TO uiEndingIndex BY 1 DO 
	IF arr_usiRecipeSetting[uiRecipeInvertIter] = 0 THEN
		arr_usiRecipeSetting[uiRecipeInvertIter]	:= 255;
	ELSIF arr_usiRecipeSetting[uiRecipeInvertIter] <> 0 THEN
		arr_usiRecipeSetting[uiRecipeInvertIter]	:= 0;
	END_IF
END_FOR

iInvertRecipeSM		:= 20;

20:
IF NOT R_TInvertRecipe.Q THEN
	iInvertRecipeSM		:= 0;
END_IF

END_CASE
END_ACTION

ACTION SeqTestMotor:

END_ACTION

ACTION SeqTestOnce:
//Run Once - DMX Channels only for now

rt_RunSeqTestOnce();
rt_ResetTestSeq();

CASE iCompareSeq[ENUM_SeqSM.Once] OF
	
0: // If test is triggered by user
//Trigger should be something like 
IF rt_RunSeqTestOnce.Q THEN
	xDMXSeqTestInProgressOnce				:= TRUE;
	uiLoopRcvIndex							:= cuiMinDUTIndex; 
	iCompareSeq[ENUM_SeqSM.Once]			:= 10;
END_IF

10: // Zero out all comparison buffers before each comparison
IF (uiLoopRcvIndex=0) THEN
	IF xDMXSeqTestInProgressOnce THEN
//by default, Counter = 0 at the first initialization; it is reset at the end of this State Machine
//Clear Storage Buffers pre-test to ensure no old data interferes with current test
		FOR uiCounter4 := 0 TO gc.uiMaxNrDMXTestCh BY 1 DO
			arrxExpctdTmpPNPSeqDMX[uiCounter4]		:= 0;		//should be all 0s ; PNP<>DMX
			arrxExpctdTmpNPNSeqDMX[uiCounter4]		:= 0;
//			arrxExpctdTmpPNPSeqDC[uiCounter4]		:= 0;		
//			arrxExpctdTmpNPNSeqDC[uiCounter4]		:= 0;
			arrxRcvdBufferPNPSeq[uiCounter4]		:= 0;		//should be all 0s too ; PNP<>DMX	
			arrxRcvdBufferNPNSeq[uiCounter4]		:= 0;
			gFB.arrFB_DMX[uiCounter4].I.xCmdOff	:= TRUE;				
		END_FOR
	iCompareSeq[ENUM_SeqSM.Once]					:= 20;
	END_IF
ELSIF (uiLoopRcvIndex>0) THEN // to avoid 
	IF xDMXSeqTestInProgressOnce AND tonTestIterGap.Q THEN
		tonTestIterGap.IN	:= FALSE;
		//by default, Counter = 0 at the first initialization; it is reset at the end of this State Machine
		//Clear Storage Buffers pre-test to ensure no old data interferes with current test
		FOR uiCounter4 := 0 TO gc.uiMaxNrDMXTestCh BY 1 DO
			arrxExpctdTmpPNPSeqDMX[uiCounter4]		:= 0;		//should be all 0s - PNP<>DMX
			arrxExpctdTmpNPNSeqDMX[uiCounter4]		:= 0;
			arrxRcvdBufferPNPSeq[uiCounter4]		:= 0;		
			arrxRcvdBufferNPNSeq[uiCounter4]		:= 0;
		END_FOR
		
	iCompareSeq[ENUM_SeqSM.Once]					:= 20; // don't write the hardware value (skip 20)
	END_IF	
END_IF
	
20:	
//write 'hardware-clear' state 
g_ast.DMXHWOut									:= g_ast.DMXPhysOut;

iCompareSeq[ENUM_SeqSM.Once]					:= 25;

25:
//Copy static test indices from Expected_Static - as these should still be used for comparisons
//	IF (arrui24VTestIndices[uiCounter4] <> 0) THEN	
//		MEMCPY(srcAddr:=ADR(arrxExpctdTmpPNP24V[cuiMinDUTIndex]),destAddr:=ADR(arrxExpctdTmpPNPSeqDMX[cuiMinDUTIndex]),n:=gc.uiChannelsUT);
FOR uiCounter4 := 0 TO gc.uiMaxNrDMXTestCh BY 1 DO
	arrxExpctdTmpPNPSeqDMX[uiCounter4]		:= arrxExpctdTmpPNP24V[uiCounter4];
	arrxExpctdTmpNPNSeqDMX[uiCounter4]		:= arrxExpctdTmpNPNGND[uiCounter4];
END_FOR

iCompareSeq[ENUM_SeqSM.Once]					:= 30;

30: //Set the Expected Mask & write data to controller
//Write the first index from the specified array of indices
//MEMCPY(srcAddr:=ADR(arrxExpctdTmpNPN[arruiSeqTestIndicesDMX[uiLoopRcvIndex]]),destAddr:=ADR(arrxExpctdTmpNPNSeqDMX[arruiSeqTestIndicesDMX[uiLoopRcvIndex]]),n:=SIZEOF(arrxExpctdTmpNPN[arruiSeqTestIndicesDMX[uiLoopRcvIndex]]));	

//This line copies only the value of the current iterator's index in the DMX Channel Array
arrxExpctdTmpNPNSeqDMX[uiLoopRcvIndex]	:= arrxExpctdTmpNPN[uiLoopRcvIndex];

iCompareSeq[ENUM_SeqSM.Once]			:= 35;

35:
IF (arruiSeqTestIndicesDMXSW[uiLoopRcvIndex] <> 0) THEN
//Also copy this specific channel index value to the comparison array
	
//Don't copy PNP indices for DMX; this doesn't generally make sense
//	MEMCPY(srcAddr:=ADR(arrxExpctdTmpPNP[arruiSeqTestIndicesDMX[uiLoopRcvIndex]]),destAddr:=ADR(arrxExpctdTmpPNPSeqDMX[arruiSeqTestIndicesDMX[uiLoopRcvIndex]]),n:=1);
	
	//CmdOn - command on - that respective channel
	gFB.arrFB_DMX[arruiSeqTestIndicesDMXSW[uiLoopRcvIndex]].I.xCmdOn			:= TRUE;
	//and turn off all others
	FOR uiCounter3 := cuiMinDUTIndex TO gc.uiMaxNrDMXTestCh BY 1 DO
		IF uiCounter3 <> arruiSeqTestIndicesDMXSW[uiLoopRcvIndex] THEN
			gFB.arrFB_DMX[uiCounter3].I.xCmdOff	:= TRUE;	
		END_IF
	END_FOR
END_IF

iCompareSeq[ENUM_SeqSM.Once]		:= 40;

40:
//Write to hardware
g_ast.DMXHWOut							:= g_ast.DMXPhysOut;
//tonWriteCopyWait.IN						:= TRUE;
iCompareSeq[ENUM_SeqSM.Once]			:=	60;

(*
50:

//Timer marks end of sampling period; reset timer
IF tonWriteCopyWait.Q THEN
	tonWriteCopyWait.IN					:=	FALSE;
	iCompareSeq[ENUM_SeqSM.Once]		:=	60;
END_IF
*)

60:
//Log all the 'gates' - returned from FB_Debounce
FOR uiCounter3	:= 0 TO gc.uiMaxNrDMXTestCh BY 1 DO
	arrxRcvdBufferNPNSeq[uiCounter3]		:= g_ast.arrFBIntNPN[uiCounter3].Q.xGate;
END_FOR
	
iCompareSeq[ENUM_SeqSM.Once]		:=	70;

//IF tonReadWait.Q THEN
//	tonReadWait.IN					:= FALSE;
//Copy hardware state
//	arrxRcvdBufferNPNSeq			:= arrxTestChInputNPN; // linked to hardware
//	arrxRcvdBufferPNPSeq			:= arrxTestChInputPNP; // linked to hardware
//iCompareSeq[ENUM_SeqSM.Once]		:= 90;
//END_IF

70:
//Run Comparos
//Individual
arr_diTestNPNSeqOnceLine[uiLoopRcvIndex]			:= MEMCMP(pBuf1:=ADR(arrxExpctdTmpNPNSeqDMX[uiLoopRcvIndex]),pBuf2:=ADR(arrxRcvdBufferNPNSeq[uiLoopRcvIndex]),n:=SIZEOF(arrxExpctdTmpNPNSeqDMX[uiLoopRcvIndex])); 
//Complete Buffer
arrdiTestNPNSeqOnceComplete[uiLoopRcvIndex]			:= MEMCMP(pBuf1:=ADR(arrxExpctdTmpNPNSeqDMX[cuiMinDUTIndex]),pBuf2:=ADR(arrxRcvdBufferNPNSeq[cuiMinDUTIndex]),n:=gc.uiChannelsUT); 

//log the error index - later

iCompareSeq[ENUM_SeqSM.Once]				:= 80;

80: //Turn off all DMX channels after comparison
FOR uiCounter3 := cuiMinDUTIndex TO gc.uiMaxNrDMXTestCh BY 1 DO
	gFB.arrFB_DMX[uiCounter3].I.xCmdOff		:= TRUE;
END_FOR

90://Write to DMX hardware, advance state
g_ast.DMXHWOut								:= g_ast.DMXPhysOut;

iCompareSeq[ENUM_SeqSM.Once]				:= 100;

100: //Confirm 'return' to static 
FOR uiCounter3	:= 0 TO gc.uiMaxNrDMXTestCh BY 1 DO
	arrxRcvdBufferNPNSeq[uiCounter3]		:= g_ast.arrFBIntNPN[uiCounter3].Q.xGate;
	IF arrxRcvdBufferNPNSeq[uiCounter3] = arrxExpctdTmpNPNGND[uiCounter3] THEN
		iCompareSeq[ENUM_SeqSM.Once]				:= 110;
	END_IF
END_FOR

110://Write to DMX hardware, advance state
g_ast.DMXHWOut								:= g_ast.DMXPhysOut;

iCompareSeq[ENUM_SeqSM.Once]				:= 120;

120: // If counter is equal to the max # of test channels, reset it; else, proceed around again 
IF (uiLoopRcvIndex = gc.uiMaxNrDMXTestCh) THEN
	iCompareSeq[ENUM_SeqSM.Once]			:= 130;
ELSE
	uiLoopRcvIndex							:= uiLoopRcvIndex +1;
	//Next iteration
	tonTestIterGap.IN						:= TRUE;
	iCompareSeq[ENUM_SeqSM.Once]			:= 10;
 (*iCounter <> gc.usiMaxNrOfChannels*)
END_IF

130:
xDMXSeqTestInProgressOnce					:= FALSE;
iCompareSeq[ENUM_SeqSM.Once]				:= 140;

140:
IF rt_ResetTestSeq.Q AND NOT rt_RunSeqTestOnce.Q THEN
	FOR uiCounter2 := 0 TO gc.uiMaxNrDMXTestCh BY 1 DO 
		arr_diTestPNPSeqOnceLine[uiCounter2]		:= 0;
		arr_diTestNPNSeqOnceLine[uiCounter2]		:= 0;
//		arrdiTestPNPSeqOnceComplete[uiCounter2]		:= 0;
//		arrdiTestNPNSeqOnceComplete[uiCounter2]		:= 0;
		arrdiTestNPNSeqOnceCompleteProblemIndex[uiCounter2]	:= 0;
	END_FOR
	diCompTestResult							:= 0;
	iCompareSeq[ENUM_SeqSM.Once]				:= 0; (* reset to beginning *)
END_IF

END_CASE
END_ACTION

ACTION SeqTestOnceDC:

END_ACTION

END_PROGRAM

(* stored: Version 1.1.0.1, ProductVersion 3.1.4024.9
   POU DMXTest: Id {56d10ee8-0ed5-46cc-a7ec-34100a2134e6}, SpecialFunc None
   Action InvertRecipeSettings: Id {ab56e97d-bd56-40c0-9de3-e9e4dcae7cf6}
   Action SeqTestMotor: Id {8ebcdac7-001b-4114-a17b-b08d6ad9551b}
   Action SeqTestOnce: Id {da9d395e-68b9-4202-9635-b7973c50d5fe}
   Action SeqTestOnceDC: Id {a6580177-07fa-4403-b780-55710f1004e3} *)
